(* Schneider Machine Expert - Basic project timer test, file version 1.6.0.0 *)
(* ProjectInformations: Name=New project *)

HARDWARE
  Cpu 0: TM221CE16R
  EthernetConfiguration: NetworkName=M221, IpAllocationMode=FixedAddress, IpAddress=0.0.0.0, SubnetMask=0.0.0.0
  SerialLineConfiguration: Baud=Baud19200, Parity=ParityEven, DataBits=DataBits8, StopBits=StopBits1, PhysicalMedium=PhysicalMediumRs485, TransmissionMode=TransmissionModeModbusRtu, SlaveId=1, Addressing=SlaveAddressing
  MastTask: UsePeriodScanMode=false, PeriodScan=100
  FastTask: Period=255
  CpuBehavior: StartingMode=StartAsPreviousState, AutoSaveRamOnEeprom=true, WatchdogPeriod=250

SYMBOLS  (address, symbol, comment, settings)

POU New POU
  (* SectionNumber=0 *)

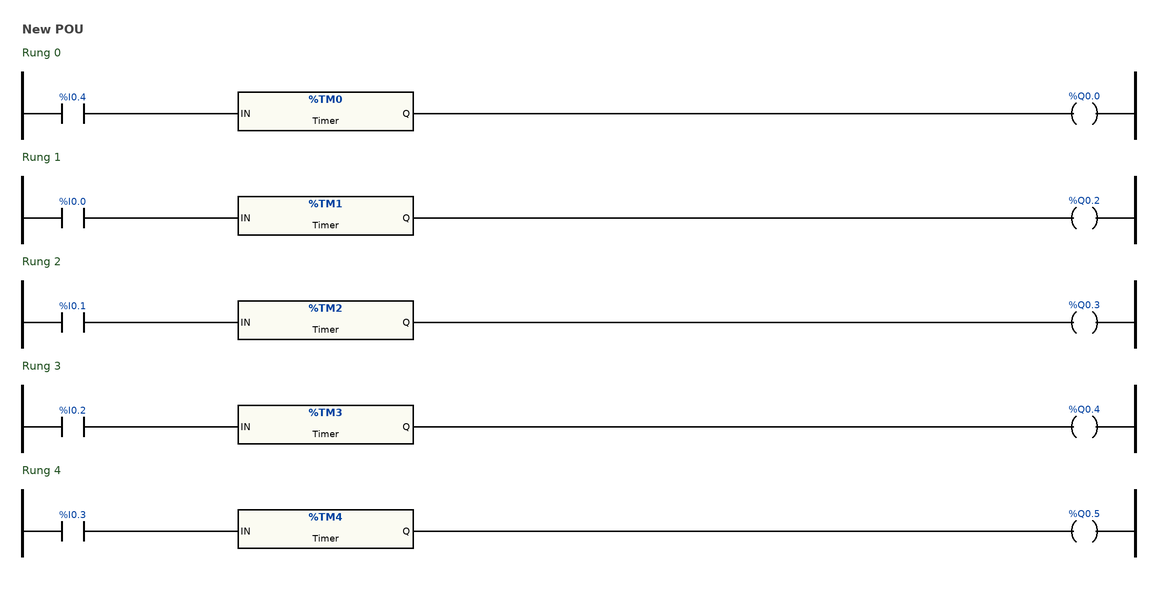

// Rung 0
  BLK %TM0
  LD %I0.4
  IN
  OUT_BLK
  LD Q
  ST %Q0.0
  END_BLK
  // as ST:
  //   %TM0(IN := %I0.4);
  //   %Q0.0 := %TM0.Q;

// Rung 1
  BLK %TM1
  LD %I0.0
  IN
  OUT_BLK
  LD Q
  ST %Q0.2
  END_BLK
  // as ST:
  //   %TM1(IN := %I0.0);
  //   %Q0.2 := %TM1.Q;

// Rung 2
  BLK %TM2
  LD %I0.1
  IN
  OUT_BLK
  LD Q
  ST %Q0.3
  END_BLK
  // as ST:
  //   %TM2(IN := %I0.1);
  //   %Q0.3 := %TM2.Q;

// Rung 3
  BLK %TM3
  LD %I0.2
  IN
  OUT_BLK
  LD Q
  ST %Q0.4
  END_BLK
  // as ST:
  //   %TM3(IN := %I0.2);
  //   %Q0.4 := %TM3.Q;

// Rung 4
  BLK %TM4
  LD %I0.3
  IN
  OUT_BLK
  LD Q
  ST %Q0.5
  END_BLK
  // as ST:
  //   %TM4(IN := %I0.3);
  //   %Q0.5 := %TM4.Q;
